(* PLC project PLC_ODOT.project, CODESYS CODESYS V3.5 SP19 *)
(* stored: creationDateTime 2026-01-26T16:59:36.3702007, modificationDateTime 2026-01-26T16:51:59.9229809 *)

FUNCTION_BLOCK FbBlink
  VAR_INPUT
    TimeOn : DINT := 2000;  (* Время включения лампочки [мс]. *)
    TimeOff : DINT := 2000;  (* Время выключения лампочки [мс]. *)
    Ts_ms : DINT := 100;  (* Шаг дискретизации по времени [мс]. *)
    Reset : BOOL := FALSE;  (* Сброс при перезагрузке. *)
  END_VAR
  VAR_OUTPUT
    BlinkLamp : BOOL := FALSE;  (* Мигающая лампочка. *)
  END_VAR
  VAR
    Timer1 : DINT := 0;  (* Таймер1 [мс]. *)
    State1 : INT := 0;  (* Граф состояний. *)
  END_VAR
  VAR CONSTANT
    STATE_RESET : INT := 0;  (* Константы. *)
    STATE_ON : INT := 1;
    STATE_OFF : INT := 2;
  END_VAR

            //            DbBlink 
//    +---------------------+
//    |       FbBlink       |
//   -|TimeOn      BlinkLamp|->-
//   -|TimeOff              |
//   -|Ts_ms                |
//   -|Reset                |
//    +---------------------+

//Пример построения универсального кроссплатформенного графа состояний.
//Использую этот код как заготовку под более сложные алгоритмы.
//Данный алгоритм гораздо быстрее разрабатывать чем конечный автомат с памятьтю.

IF (Reset) THEN //Сброс при перезагрузке.
State1 := STATE_RESET;
END_IF;

CASE (State1) OF //Граф состояний.

STATE_RESET: //Сброс.
BlinkLamp := FALSE;
Timer1    := 0;
State1 := STATE_ON;

STATE_ON: //Включить лампочку на заданное время.
BlinkLamp := TRUE;
Timer1 := Timer1 + Ts_ms;
IF (Timer1 >= TimeOn) THEN
State1 := STATE_OFF;
Timer1 := 0;
END_IF;    

STATE_OFF: //Выключить лампочку на заданное время.
BlinkLamp := FALSE;
Timer1 := Timer1 + Ts_ms;
IF (Timer1 >= TimeOff) THEN
State1 := STATE_ON;
Timer1 := 0;
END_IF;    

ELSE //RESET при неопределенном состоянии.
State1 := STATE_RESET;
END_CASE; //CASE (State1) OF

// Граф состояний.
//
//            |
//           -+- Reset
//            |
//            V
//  +-------------------+
//  | State1 =          |
//  | STATE_RESET       |
//  | BlinkLamp = 0     |
//  +-------------------+
//            |
//            |
//            |
//            |
//            V
//  +-------------------+
//  | State1 =          |
//  | STATE_ON          |<--------------+
//  | BlinkLamp = 1     |               |
//  +-------------------+               |
//            |                         |
//            |                         |
//           -+- Timer1 >= TimeOn      -+- Timer1 >= TimeOff
//            |                         |
//            V                         |
//  +-------------------+               |
//  | State1 =          |               |
//  | STATE_OFF         |---------------+
//  | BlinkLamp = 0     |
//  +-------------------+

//  +---------+
//  | GNU GPL |
//  +---------+
//  |
//  |
//  .= .-_-. =.
// ((_/)o o(\_))
//  `-'(. .)`-'
//  |/| \_/ |\
//  ( |     | )
//  /"\_____/"\
//  \__)   (__/
// @COPYLEFT ALL WRONGS RESERVED :)
// Author: VA
// Contacts: DIY.PLC.314@gmail.com
// License: GNU GPL v2
//
// https://www.youtube.com/@DIY_PLC
// https://github.com/DIYPLC

          
END_FUNCTION_BLOCK
